{attribute addProperty BoxType "AT2050-0501-0023"}
{attribute addProperty Id "A_0083_AT2050_5500_0016_AT2050_5500AT2050_3DCFC8D064080"}
{attribute addProperty CRC "426597251"}
{attribute addProperty SizeInBites "640"}
{attribute addProperty SizeInBytes "80"}
TYPE A_0071_AT2050_0501_0023_AT2050_0501_196D5B83 EXTENDS AT2050_9506A482 :
STRUCT
	{attribute addProperty Name "A_0083_AT2050_5500_0016_AT2050_5500"}
	A_0083_AT2050_5500_0016_AT2050_5500 : AT2050_3DCFC8D0;
END_STRUCT
END_TYPE

(* stored: Version 1.2.0.0, ProductVersion 3.1.4024.9
   DUT A_0071_AT2050_0501_0023_AT2050_0501_196D5B83: Id {e6e8905a-3a5e-4ddd-b171-a31631fd30eb} *)
